(* IEC 61131-3 sources: Industry-PLC-LLM/data/PLCBEAD_repo/PLCBEAD_PLCEmbed-main/PLC-BEAD/Source/GEB/CONTROL_SET1, 1 file *)

(* ---- CONTROL_SET1.ST ---- *)
FUNCTION_BLOCK CONTROL_SET1_Block
	VAR_INPUT
		KT :	REAL;
		TT :	REAL;
		PI :	BOOL;
		PIDD :	BOOL;
		P_K :	REAL := 0.5;
		PI_K :	REAL := 0.45;
		PI_TN :	REAL := 0.83;
		PIDD_K :	REAL := 0.6;
		PIDD_TN :	REAL := 0.5;
		PIDD_TV :	REAL := 0.125;
	END_VAR

	VAR_OUTPUT
		KP :	REAL;
		TN :	REAL;
		TV :	REAL;
		KI :	REAL;
		KD :	REAL;
	END_VAR

	IF PI AND PIDD THEN
		KP := 0.0;
		TN := 0.0;
		TV := 0.0;
	ELSIF PIDD THEN
		KP := PIDD_K * KT;
		TN := PIDD_TN * TT;
		TV := PIDD_TV * TT;
	ELSIF PI THEN
		KP := PI_K * KT;
		TN := PI_TN * TT;
	ELSE
		KP := P_K * KT;
	END_IF;
	IF TN > 0.0 THEN KI := KP / TN; ELSE KI := 0.0; END_IF;
	KD := KP * TV;
END_FUNCTION_BLOCK

PROGRAM program0
  VAR
	KT :REAL;
	TT :REAL;
	PI :BOOL;
	PIDD :BOOL;
	P_K :REAL ;
	PI_K :REAL ;
	PI_TN :REAL ;
	PIDD_K :REAL ;
	PIDD_TN :REAL ;
	PIDD_TV :REAL ;
	KP :REAL;
	TN :REAL;
	TV :REAL;
	KI :REAL;
	KD :REAL;
	func_block : CONTROL_SET1_Block;
  END_VAR
	func_block.KT   :=KT  ;
	func_block.TT   :=TT  ;
	func_block.PI   :=PI  ;
	func_block.PIDD   :=PIDD  ;
	func_block.P_K   :=P_K  ;
	func_block.PI_K   :=PI_K  ;
	func_block.PI_TN   :=PI_TN  ;
	func_block.PIDD_K   :=PIDD_K  ;
	func_block.PIDD_TN   :=PIDD_TN  ;
	func_block.PIDD_TV   :=PIDD_TV  ;
	func_block();
	KP := func_block.KP ;
	TN := func_block.TN ;
	TV := func_block.TV ;
	KI := func_block.KI ;
	KD := func_block.KD ;
END_PROGRAM
